Staubli VAL3: remMovJoint.pgx

program remMovJoint(string& sArgs[] (dimensions=1), string& sReturn[] (dimensions=1))
  local bool bOk
  local joint jDest
  local num nLoop
  local num nVal
  local point pDest
  local string sArgsLoop
begin
  // Move to the designated point.
  //
  // Arguments are "J1 J2 J3 J4 J5 J6"
  //
  logMsg("call remMovJoint")
  //break down our 6 args and make sure they are numbers
  jDest={0,0,0,0,0,0}
  nLoop=0
  sArgsLoop=sArgs
  while nLoop<6
    sArgsLoop=toNum(sArgsLoop,nVal,bOk)
    if bOk
      switch nLoop
        case 0
          jDest.j1=nVal
        break
        case 1
          jDest.j2=nVal
        break
        case 2
          jDest.j3=nVal
        break
        case 3
          jDest.j4=nVal
        break
        case 4
          jDest.j5=nVal
        break
        case 5
          jDest.j6=nVal
        break
      endSwitch
      nLoop=nLoop+1
    else
      call remErrNum("MOVJOINT",sArgs,sReturn)
      return
    endIf
  endWhile
  if nIPNumber==0
    pDest=jointToPoint(tSensorTool,fIP1,jDest)
  else
    pDest=jointToPoint(tSensorTool,fIP2,jDest)
  endIf
  call remMovBase(pDest,sReturn)
end
